FUNCTION_BLOCK AROBOT_MUX (* Composite FB wrapping other FBs *)
  (* Standard: 61499-2 *)
  (* Version 0.0, 2008-07-10, 4DIAC-IDE, 4DIAC-Consortium *)
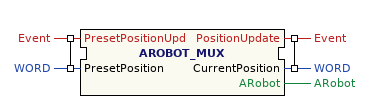
  EVENT_INPUT
    PresetPositionUpd WITH PresetPosition; (* Indication from Plug *)
  END_EVENT
  EVENT_OUTPUT
    PositionUpdate WITH CurrentPosition; (* Request from Socket *)
  END_EVENT
  VAR_INPUT
    PresetPosition : WORD; (* Confirmation Data from Plug *)
  END_VAR
  VAR_OUTPUT
    CurrentPosition : WORD; (* Request Data from Socket *)
  END_VAR
  PLUGS
    ARobot : ARobot;
  END_PLUGS
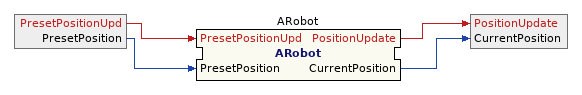
  EVENT_CONNECTIONS
    PresetPositionUpd TO ARobot.PresetPositionUpd;
    ARobot.PositionUpdate TO PositionUpdate;
  END_CONNECTIONS
  DATA_CONNECTIONS
    PresetPosition TO ARobot.PresetPosition;
    ARobot.CurrentPosition TO CurrentPosition;
  END_CONNECTIONS
END_FUNCTION_BLOCK
